FUNCTION F_PrimeCheck : BOOL
VAR_INPUT
	nInputNum : INT;
	
END_VAR

VAR
	nLimit : INT;
	nIterator : INT;
END_VAR


F_PrimeCheck := TRUE;
IF nInputNum > 1 THEN
	nLimit := nInputNum/2;
	FOR nIterator := 2 TO nLimit  DO
		IF (nInputNum MOD nIterator) = 0 THEN 
			F_PrimeCheck := FALSE;
			EXIT;
		END_IF
	END_FOR
END_IF
IF nInputNum <=1 THEN 
	F_PrimeCheck := FALSE;
	RETURN;
END_IF

END_FUNCTION

(* stored: Version 1.1.0.1, ProductVersion 3.1.4024.16
   POU F_PrimeCheck: Id {132a477c-cae7-4a95-964a-acd88e85aa3b}, SpecialFunc None *)
